Fanuc KAREL source: KD00063.KL

PROGRAM KD00063
%NOLOCKGROUP
VAR
  I: INTEGER
  J: INTEGER
  B: BOOLEAN
  R: REAL
  S: STRING[80]
BEGIN
  CONDITION[1]:
  WHEN DIN[1] = ON DO
    ENABLE CONDITION[1]
  ENDCONDITION
END KD00063
